Fanuc KAREL source: kt00381.compact.KL

PROGRAM KT00381
%STACKSIZE=65535
%PRIORITY=65535
%NOLOCKGROUP
VAR
H1 : ARRAY[2] OF SHORT
Y2 : ARRAY[2] OF BYTE
OUT : BOOLEAN
BEGIN
H1[1]=2
Y2[1]=3
OUT=(H1[1] <=Y2[1])
END KT00381
